// TIA Portal V17 export
// export: Created 2022-07-31T06:40:44.8485819Z, ExportSetting WithDefaults, DisplayName Totally Integrated Automation Portal, DisplayVersion V17 Update 2, DisplayName TIA Portal Openness, DisplayVersion V17 Update 2, DisplayName TIA Portal Version Control Interface, DisplayVersion V17, DisplayName SINAMICS Startdrive Advanced, DisplayVersion V17 Update1, DisplayName SINAMICS Startdrive G110M, G120, G120C, G120D, G120P, G115D, DisplayVersion V17 Update1, DisplayName SINAMICS Startdrive G130, G150, S120, S150, SINAMICS MV, S210, DisplayVersion V17 Update1, DisplayName STEP 7 Professional, DisplayVersion V17 Update 2, DisplayName STEP 7 Safety, DisplayVersion V17, DisplayName WinCC UA Professional, DisplayVersion V17 Update 2
DATA_BLOCK "logger"   // DB1
{ DB_Accessible_From_OPC_UA := 'FALSE' }
VERSION : 0.1
// stored: AutoNumber true, DBAccessibleFromOPCUA false, DBAccessibleFromWebserver false, InstanceOfName LoggerFb, InstanceOfType FB
"LoggerFb"
   // VAR_INPUT
   //    global_logger_level { ExternalAccessible := 'False'; ExternalVisible := 'False'; ExternalWritable := 'False'} : USInt;
   //    ip_1 { ExternalAccessible := 'False'; ExternalVisible := 'False'; ExternalWritable := 'False'} : USInt;
   //    ip_2 { ExternalAccessible := 'False'; ExternalVisible := 'False'; ExternalWritable := 'False'} : USInt;
   //    ip_3 { ExternalAccessible := 'False'; ExternalVisible := 'False'; ExternalWritable := 'False'} : USInt;
   //    ip_4 { ExternalAccessible := 'False'; ExternalVisible := 'False'; ExternalWritable := 'False'} : USInt;
   //    port_number { ExternalAccessible := 'False'; ExternalVisible := 'False'; ExternalWritable := 'False'} : UInt;
   //    interface_id { ExternalAccessible := 'False'; ExternalVisible := 'False'; ExternalWritable := 'False'} : UInt;
   //    id { ExternalAccessible := 'False'; ExternalVisible := 'False'; ExternalWritable := 'False'} : CONN_OUC;
   // END_VAR
   // VAR_OUTPUT
   //    buffer_size { ExternalAccessible := 'False'; ExternalVisible := 'False'; ExternalWritable := 'False'} : Int;
   // END_VAR
   // VAR
   //    tsend { ExternalAccessible := 'False'; ExternalVisible := 'False'; ExternalWritable := 'False'; S7_SetPoint := 'True'} : TSEND_C;
   //    connect { ExternalAccessible := 'False'; ExternalVisible := 'False'; ExternalWritable := 'False'; S7_SetPoint := 'True'} : TCON_IP_v4;
   //    data { ExternalAccessible := 'False'; ExternalVisible := 'False'; ExternalWritable := 'False'} : String;
   //    buffer { ExternalAccessible := 'False'; ExternalVisible := 'False'; ExternalWritable := 'False'} : Array[0..9] of String;
   //    state { ExternalAccessible := 'False'; ExternalVisible := 'False'; ExternalWritable := 'False'} : Int;
   //    timeout { ExternalAccessible := 'False'; ExternalVisible := 'False'; ExternalWritable := 'False'} : TON_TIME;
   //    init { ExternalAccessible := 'False'; ExternalVisible := 'False'; ExternalWritable := 'False'; S7_SetPoint := 'True'} : Bool;
   //    config_in_block { ExternalAccessible := 'False'; ExternalVisible := 'False'; ExternalWritable := 'False'} : Struct
   //       level { ExternalAccessible := 'False'; ExternalVisible := 'False'; ExternalWritable := 'False'} : USInt;
   //       block_title { ExternalAccessible := 'False'; ExternalVisible := 'False'; ExternalWritable := 'False'} : String;
   //    END_STRUCT;
   // END_VAR
BEGIN
END_DATA_BLOCK
